{attribute 'GeneratedUsingTerminal: ELM2644-0000-0016'}
{attribute addProperty BoxType "ELM2644-0000-0016"}
{attribute addProperty Id "Outputs_Channel_4AT %Q*Outputs_Channel_78994C084"}
{attribute addProperty CRC "1582630039"}
{attribute addProperty Size "4"}
TYPE DO_Group_4_Outputs_5E550497 :
STRUCT
	{attribute addProperty Name "Outputs_Channel_4"}
	Outputs_Channel_4 AT %Q* : Outputs_Channel_78994C08;
END_STRUCT
END_TYPE

(* stored: Version 1.2.0.0, ProductVersion 3.1.4024.9
   DUT DO_Group_4_Outputs_5E550497: Id {6b572a51-9d51-4c3f-a159-2327788c49dc} *)
